FUNCTION_BLOCK TONOFF
VAR_INPUT
	IN: BOOL;
	PT:TIME;
END_VAR
VAR_OUTPUT
	Q:BOOL;
END_VAR
VAR
	timeOn:TON;
	timeOff:TOF;
	state: INT;
	Timer: INT;
END_VAR

timeOn(IN:=IN,PT:=PT,Q=>,ET=>);
timeOff(In:=timeOn.Q,PT:=PT,Q=>Q,ET=>);

END_FUNCTION_BLOCK

(* stored: Version 1.1.0.1, ProductVersion 3.1.4024.11
   POU TONOFF: Id {e443702c-a28c-4830-85fc-658524f944e7}, SpecialFunc None *)
